(* CODESYS project WindaFBD.project

Project tree, tasks and I/O mapping:
  Device : CODESYS Control Win V3, 3S - Smart Software Solutions GmbH, order no. 305021, version 3.5.8.10
    application Application
      libraries: Standard, * (System)
      task MainTask (cyclic, interval t#20ms, priority 1) calls PLC_PRG
      task VISU_TASK (cyclic, interval 100 ms, priority 31) calls VisuElems.Visu_Prg
      program PLC_PRG [FBD]
      visualisation Visualization
  text list GlobalTextList
*)

// Device/Application/PLC_PRG
PROGRAM PLC_PRG
VAR
	//WARTOŚĆ PUSTA
	RESET : BOOL;
	//ZEGAR WYZNACZAJĄCY INTERWAŁY 10ms
	TL : TON;
	//ZMIENNE ODPOWIEDZIALNE ZA CZAS
	CZAS : TIME;
	CLOCK : BOOL;	
	//PRZYCISKI GÓRA/DÓŁ
	BTN_UP : BOOL;
	BTN_DOWN : BOOL;
	//STANY INFORMUJĄCE O RUCHU WINDY GÓRA/DÓŁ
	ELEV_UP : BOOL;
	ELEV_DOWN : BOOL;
	//LICZNIK IMPUSLÓW
	COUNTER : WORD;
	//INFORMACJA CZY WINDA JEST NA GÓRZE CZY NA DOLE
	IS_ELEV_UP : BOOL;
	IS_ELEV_DOWN : BOOL;
	//LICZNIK REWERSYJNY
	C1 : CTUD;
	//PRZERZUTNIKI
	RS1 : RS;
	RS2 : RS;
	//ZMIENNA PRZECHOWUJĄCE WYSOKOŚCI POSZCZEGULNYCH PIĘTER (1-5)
	FIRST_FLOOR: WORD := 100;
	SECOND_FLOOR: WORD := 200;
	THIRD_FLOOR: WORD := 300;
	FOURTH_FLOOR: WORD := 400;
	FIFTH_FLOOR: WORD := 500;
	//ZMIENNA PRZECHOWUJĄCA WARTOŚĆ AKTYWNEGO PIĘTRA
	ACTIVE_FLOOR: WORD := 5;
	//ZMIENNE POKAZUJĄCE NA KTÓRYM PIĘTRZE JEST WINDA (1-5)
	IS_1: BOOL;
	IS_2: BOOL;
	IS_3: BOOL;
	IS_4: BOOL;
	IS_5: BOOL;
	WHICH_FLOOR: BOOL;
	//PRZYCISKI PRZYWOŁUJĄCE WINDĘ NA ODPOWIEDNIE PIĘTRO
	BTN_1: BOOL;
	BTN_2: BOOL;
	BTN_3: BOOL;
	BTN_4: BOOL;
	BTN_5: BOOL; 
END_VAR
VAR // added by the converter: edge detectors and wires of the graphical bodies
    _w1, _w2, _w3, _w4 : BOOL;
END_VAR

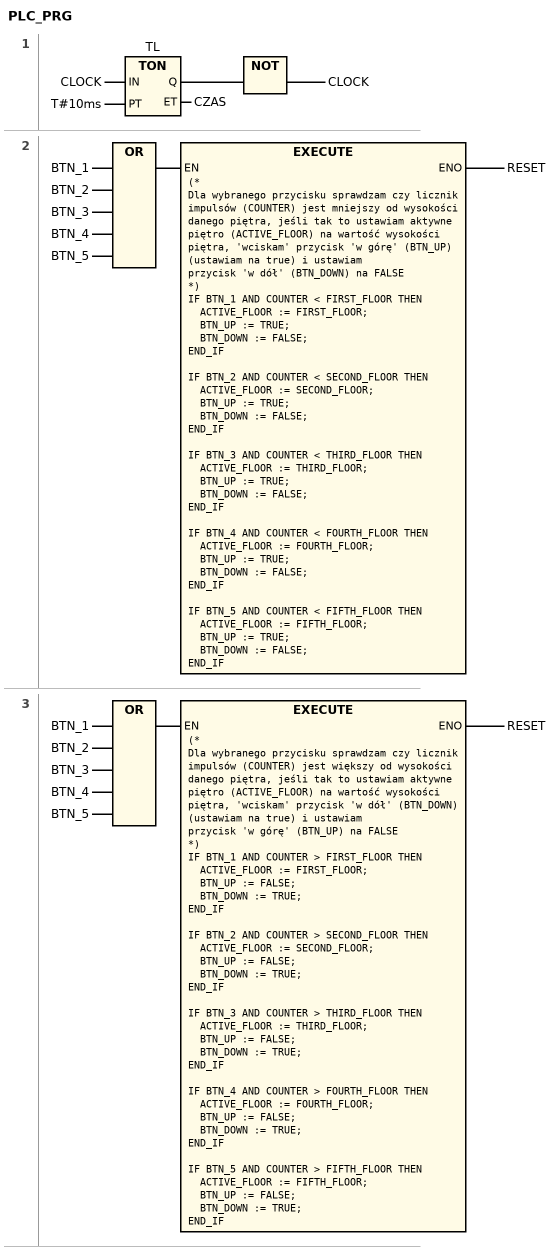
// NETWORK 1
TL(IN := CLOCK, PT := T#10ms, ET => CZAS); // TON
CLOCK := NOT TL.Q;

// NETWORK 2
_w1 := BTN_1 OR BTN_2 OR BTN_3 OR BTN_4 OR BTN_5;
IF _w1 THEN
    (*
    Dla wybranego przycisku sprawdzam czy licznik
    impulsów (COUNTER) jest mniejszy od wysokości
    danego piętra, jeśli tak to ustawiam aktywne 
    piętro (ACTIVE_FLOOR) na wartość wysokości 
    piętra, 'wciskam' przycisk 'w górę' (BTN_UP)
    (ustawiam na true) i ustawiam 
    przycisk 'w dół' (BTN_DOWN) na FALSE
    *)
    IF BTN_1 AND COUNTER < FIRST_FLOOR THEN
    	ACTIVE_FLOOR := FIRST_FLOOR;
    	BTN_UP := TRUE;
    	BTN_DOWN := FALSE;
    END_IF
    
    IF BTN_2 AND COUNTER < SECOND_FLOOR THEN
    	ACTIVE_FLOOR := SECOND_FLOOR;
    	BTN_UP := TRUE;
    	BTN_DOWN := FALSE;
    END_IF
    
    IF BTN_3 AND COUNTER < THIRD_FLOOR THEN
    	ACTIVE_FLOOR := THIRD_FLOOR;
    	BTN_UP := TRUE;
    	BTN_DOWN := FALSE;
    END_IF
    
    IF BTN_4 AND COUNTER < FOURTH_FLOOR THEN
    	ACTIVE_FLOOR := FOURTH_FLOOR;
    	BTN_UP := TRUE;
    	BTN_DOWN := FALSE;
    END_IF
    
    IF BTN_5 AND COUNTER < FIFTH_FLOOR THEN
    	ACTIVE_FLOOR := FIFTH_FLOOR;
    	BTN_UP := TRUE;
    	BTN_DOWN := FALSE;
    END_IF
END_IF
RESET := _w1;

// NETWORK 3
_w2 := BTN_1 OR BTN_2 OR BTN_3 OR BTN_4 OR BTN_5;
IF _w2 THEN
    (*
    Dla wybranego przycisku sprawdzam czy licznik
    impulsów (COUNTER) jest większy od wysokości
    danego piętra, jeśli tak to ustawiam aktywne 
    piętro (ACTIVE_FLOOR) na wartość wysokości 
    piętra, 'wciskam' przycisk 'w dół' (BTN_DOWN)
    (ustawiam na true) i ustawiam 
    przycisk 'w górę' (BTN_UP) na FALSE
    *)
    IF BTN_1 AND COUNTER > FIRST_FLOOR THEN
    	ACTIVE_FLOOR := FIRST_FLOOR;
    	BTN_UP := FALSE;
    	BTN_DOWN := TRUE;
    END_IF
    
    IF BTN_2 AND COUNTER > SECOND_FLOOR THEN
    	ACTIVE_FLOOR := SECOND_FLOOR;
    	BTN_UP := FALSE;
    	BTN_DOWN := TRUE;
    END_IF
    
    IF BTN_3 AND COUNTER > THIRD_FLOOR THEN
    	ACTIVE_FLOOR := THIRD_FLOOR;
    	BTN_UP := FALSE;
    	BTN_DOWN := TRUE;
    END_IF
    
    IF BTN_4 AND COUNTER > FOURTH_FLOOR THEN
    	ACTIVE_FLOOR := FOURTH_FLOOR;
    	BTN_UP := FALSE;
    	BTN_DOWN := TRUE;
    END_IF
    
    IF BTN_5 AND COUNTER > FIFTH_FLOOR THEN
    	ACTIVE_FLOOR := FIFTH_FLOOR;
    	BTN_UP := FALSE;
    	BTN_DOWN := TRUE;
    END_IF
END_IF
RESET := _w2;

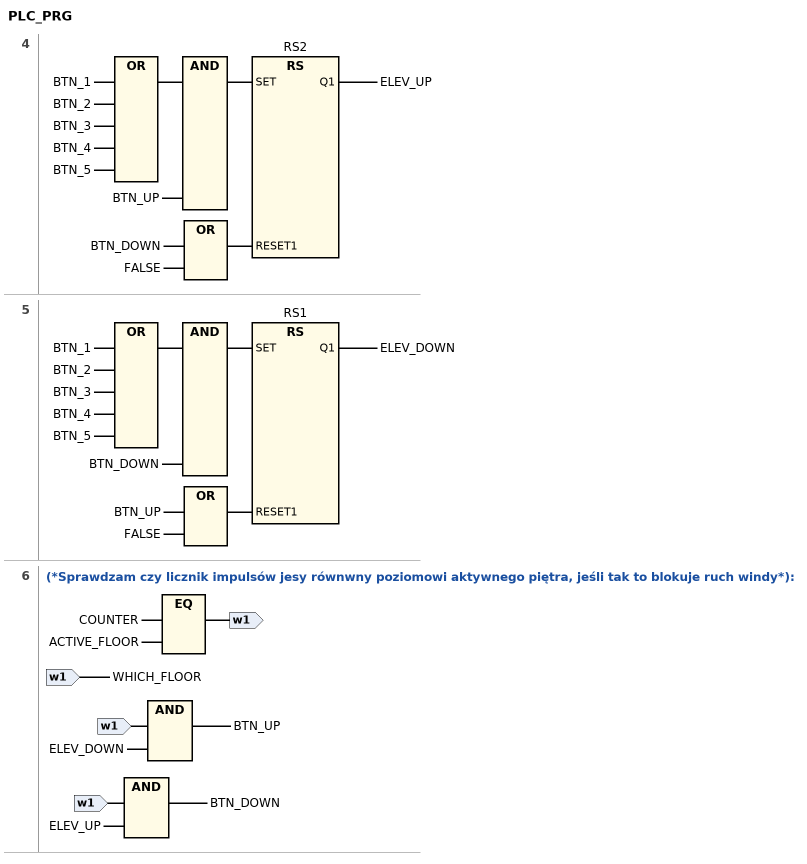
// NETWORK 4
RS2(SET := (BTN_1 OR BTN_2 OR BTN_3 OR BTN_4 OR BTN_5) AND BTN_UP, RESET1 := BTN_DOWN OR FALSE); // RS
ELEV_UP := RS2.Q1;

// NETWORK 5
RS1(SET := (BTN_1 OR BTN_2 OR BTN_3 OR BTN_4 OR BTN_5) AND BTN_DOWN, RESET1 := BTN_UP OR FALSE); // RS
ELEV_DOWN := RS1.Q1;

// NETWORK 6
// label: (*Sprawdzam czy licznik impulsów jesy równwny poziomowi aktywnego piętra, jeśli tak to blokuje ruch windy*)
_w3 := COUNTER = ACTIVE_FLOOR;
WHICH_FLOOR := _w3;
BTN_UP := _w3 AND ELEV_DOWN;
BTN_DOWN := _w3 AND ELEV_UP;

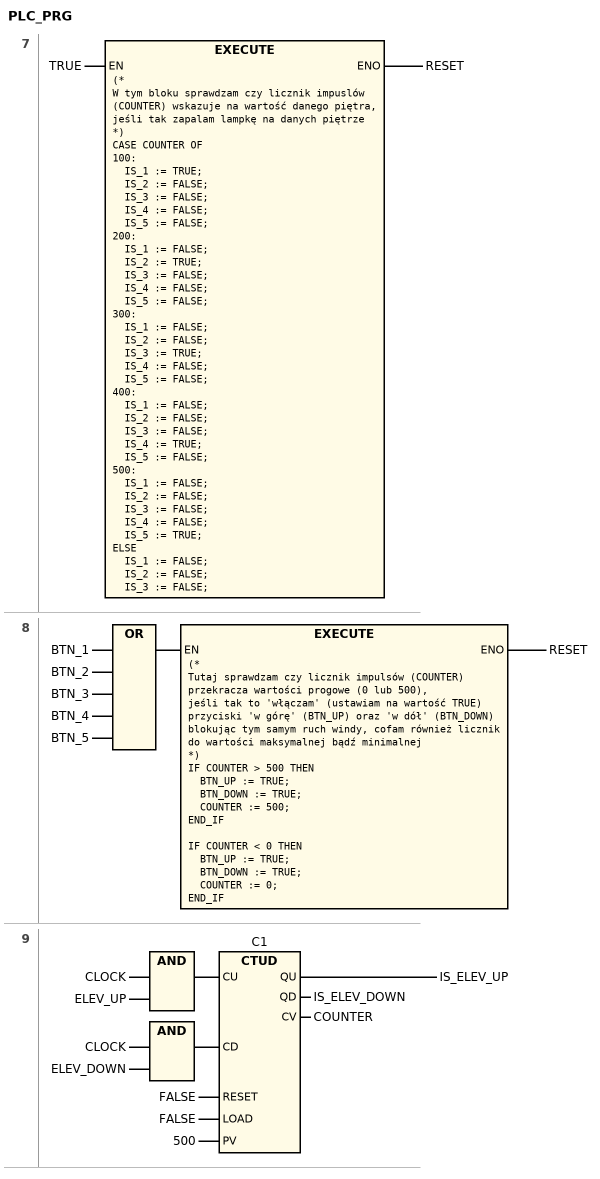
// NETWORK 7
(*
W tym bloku sprawdzam czy licznik impuslów
(COUNTER) wskazuje na wartość danego piętra,
jeśli tak zapalam lampkę na danych piętrze
*)
CASE COUNTER OF
100:
	IS_1 := TRUE;
	IS_2 := FALSE;
	IS_3 := FALSE;
	IS_4 := FALSE;
	IS_5 := FALSE;
200:
	IS_1 := FALSE;
	IS_2 := TRUE;
	IS_3 := FALSE;
	IS_4 := FALSE;
	IS_5 := FALSE;
300:
	IS_1 := FALSE;
	IS_2 := FALSE;
	IS_3 := TRUE;
	IS_4 := FALSE;
	IS_5 := FALSE;
400:
	IS_1 := FALSE;
	IS_2 := FALSE;
	IS_3 := FALSE;
	IS_4 := TRUE;
	IS_5 := FALSE;
500:
	IS_1 := FALSE;
	IS_2 := FALSE;
	IS_3 := FALSE;
	IS_4 := FALSE;
	IS_5 := TRUE;
ELSE
	IS_1 := FALSE;
	IS_2 := FALSE;
	IS_3 := FALSE;
	IS_4 := FALSE;
	IS_5 := FALSE;
END_CASE
RESET := TRUE;

// NETWORK 8
_w4 := BTN_1 OR BTN_2 OR BTN_3 OR BTN_4 OR BTN_5;
IF _w4 THEN
    (*
    Tutaj sprawdzam czy licznik impulsów (COUNTER)
    przekracza wartości progowe (0 lub 500),
    jeśli tak to 'włączam' (ustawiam na wartość TRUE) 
    przyciski 'w górę' (BTN_UP) oraz 'w dół' (BTN_DOWN)
    blokując tym samym ruch windy, cofam również licznik
    do wartości maksymalnej bądź minimalnej
    *)
    IF COUNTER > 500 THEN
    	BTN_UP := TRUE;
    	BTN_DOWN := TRUE;
    	COUNTER := 500;
    END_IF
    
    IF COUNTER < 0 THEN
    	BTN_UP := TRUE;
    	BTN_DOWN := TRUE;
    	COUNTER := 0;
    END_IF
END_IF
RESET := _w4;

// NETWORK 9
C1(
    CU := CLOCK AND ELEV_UP,
    CD := CLOCK AND ELEV_DOWN,
    RESET := FALSE,
    LOAD := FALSE,
    PV := 500,
    QD => IS_ELEV_DOWN,
    CV => COUNTER); // CTUD
IS_ELEV_UP := C1.QU;

END_PROGRAM

// Device/Application/Visualization
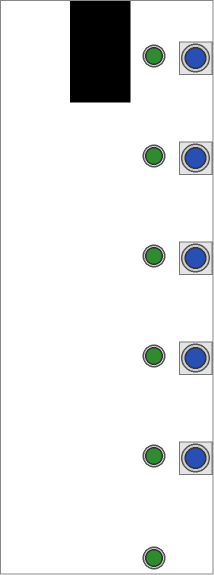
VISUALIZATION Visualization  // 214x575
    Rectangle (70,0 60x102)
        p2738717112: 500-PLC_PRG.COUNTER
    Lamp1 (141,41 26x30), variable: PLC_PRG.IS_5, style: Lamp-Lamp1-Green
    Lamp1 (141,441 26x30), variable: PLC_PRG.IS_1, style: Lamp-Lamp1-Green
    Lamp1 (141,341 26x30), variable: PLC_PRG.IS_2, style: Lamp-Lamp1-Green
    Lamp1 (141,241 26x30), variable: PLC_PRG.IS_3, style: Lamp-Lamp1-Green
    Lamp1 (141,141 26x30), variable: PLC_PRG.IS_4, style: Lamp-Lamp1-Green
    Lamp1 (141,543 26x30), variable: PLC_PRG.IS_ELEV_DOWN, style: Lamp-Lamp1-Green
    PushSwitch (179,441 33x34), variable: PLC_PRG.BTN_1, behaviour: TAP, style: Switch-PushSwitch-Blue
    PushSwitch (179,341 33x34), variable: PLC_PRG.BTN_2, behaviour: TAP, style: Switch-PushSwitch-Blue
    PushSwitch (179,241 33x34), variable: PLC_PRG.BTN_3, behaviour: TAP, style: Switch-PushSwitch-Blue
    PushSwitch (179,141 33x34), variable: PLC_PRG.BTN_4, behaviour: TAP, style: Switch-PushSwitch-Blue
    PushSwitch (179,41 33x34), variable: PLC_PRG.BTN_5, behaviour: TAP, style: Switch-PushSwitch-Blue
END_VISUALIZATION
